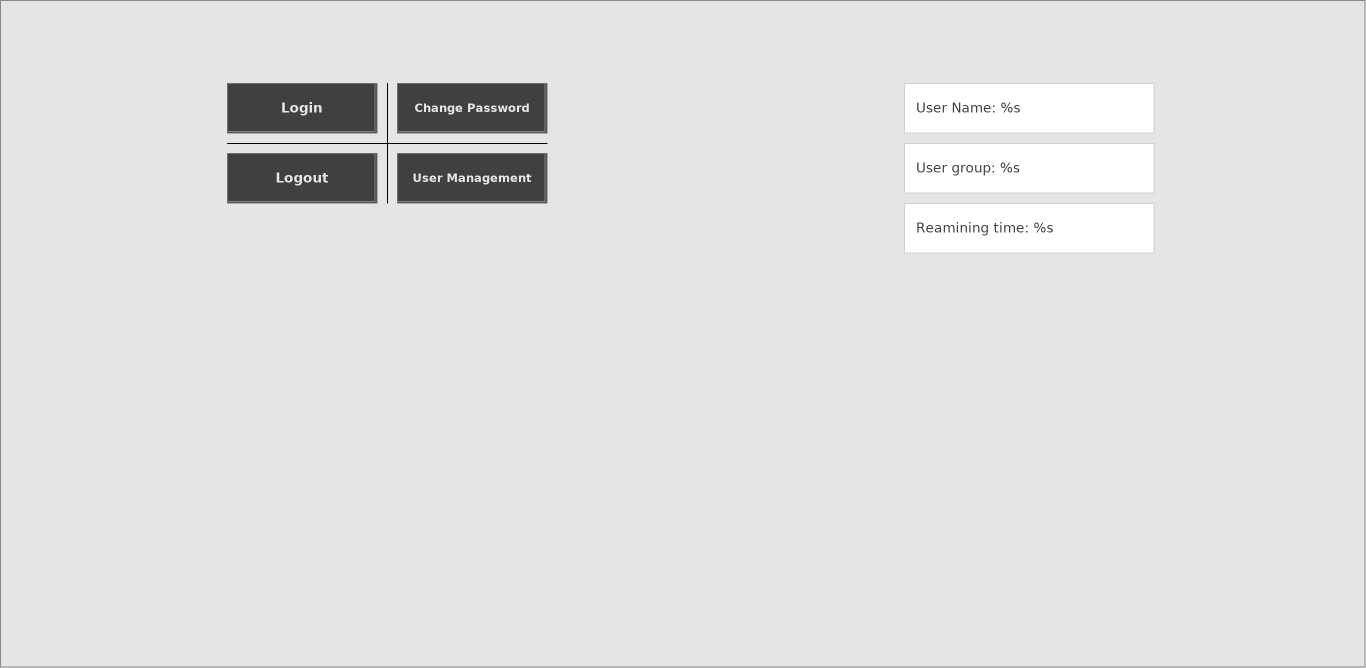
VISUALIZATION V_Users  // 1366x668
    Button (227,83 150x50), "Login"
        OnMouseDown: VisuUserMgmt Type=Login
    Button (227,153 150x50), "Logout"
        OnMouseDown: VisuUserMgmt Type=Logout
    Button (397,83 150x50), "Change Password"
        OnMouseDown: VisuUserMgmt Type=ChangeUserPassword
    Button (397,153 150x50), "User Management"
        OnMouseDown: VisuUserMgmt Type=OpenUserConfiguration
    Line (387,83) (387,203)
    Line (227,143) (547,143)
    Textfield (904,83 250x50), "User Name: %s", text variable: VisuElemsWinControls.CurrentUserName
    Textfield (904,143 250x50), "User group: %s", text variable: VisuElemsWinControls.CurrentUserGroupName
    Textfield (904,203 250x50), "Reamining time: %s", text variable: P_UserControl.sTime
END_VISUALIZATION

(* stored: Version 1.1.0.1, ProductVersion 3.1.4024.3
   Visu V_Users: Id {e2f909db-b1eb-4307-bd08-f61cc34f3330} *)
